// TIA Portal V18 export
FUNCTION_BLOCK "Capping_Station"   // FB1, LAD
TITLE = Description
{ S7_Optimized_Access := 'TRUE' }
VERSION : 0.1
// How to control and set capping station:
// 1) Start the machine
// 2) Use jog pos/neg in the capping station data block to rotate motor to read max and min value: ReadSensorMax and Read SensorMin. Based on these values update "SensorPosValMax..." and "SensorPosValMin..."
// 3) Move capping station using "MovingUP" and "MovingDOWN". The mechanism should stop top or bottom and confirm it with the change of the status "CSPositionUP" and "CSPositionDOWN". If it is constantly moving, it means that the value was not reached (too low for SensorPosValMin or too high for "SensorPosValMax").
// 
// IMPORTANT:
// - assembly of the mechanism needs to be the same, especially the position of the sensor
// - power supply for the sensor should be set to the exact voltage (5V) to provide repeteable readings
// 
// Things to implement:
// - Change sensor for limit switch
// - Improve mechanical design
// 
// E-STOP - always check!
// stored: AutoNumber true, IsIECCheckEnabled false, IsRetainMemResEnabled false, MemoryReserve 100, SetENOAutomatically false, UDAEnableTagReadback false
   VAR_INPUT
      ESTOP : Bool;
      SerialNumber : Int;
      CappingOption : Int;   // Send 1 to skip capping station
      MachineStart : Bool;
      CappingSensor : UInt;
      JogPOS : Bool;
      JogNEG : Bool;
      MoveRel : Bool;
      AxisXNotMoving : Bool;
      AxisYNotMoving : Bool;
      DoorSensor : Bool;
   END_VAR
   VAR_OUTPUT
      MovingUP : Bool;
      MovingDOWN : Bool;
      CSPositionUP : Bool;
      CSPositionDOWN : Bool;
      CSXYMotionLock : Bool;
      CappingPosition : UInt;
      MaintenanceNeeded : Bool;
   END_VAR
   VAR_IN_OUT
      CSMoveUP : Bool;
      CSMoveDOWN : Bool;
   END_VAR
   VAR
      MotionLockInternal : Bool;
      TimeSafety : Bool;
      SensorConversion : Real;
      SensorPosValMaxTrigger : UInt;
      SensorPosValMinTrigger : UInt;
      ReadSensorMax : UInt;   // Use jogging to read initial limit values
      ReadSensorMin : UInt := 10000;   // Use jogging to read initial limit values
      CountSinceON : DInt;
   END_VAR
   VAR RETAIN
      CountSinceNEW : DInt;
   END_VAR
   VAR
      MaintenanceMotionLockDisabled : Bool := true;
      SensorPosValMin { ExternalAccessible := 'False'; ExternalVisible := 'False'; ExternalWritable := 'False'} : UInt;   // 0; 14000; Machine 2009: 9000
      SensorPosValMax { ExternalAccessible := 'False'; ExternalVisible := 'False'; ExternalWritable := 'False'} : UInt;   // 6000; 21000; Machine 2009: 24500
      ScaleRangeMin { ExternalAccessible := 'False'; ExternalVisible := 'False'; ExternalWritable := 'False'} : UInt;   // 2009: 26000; 2008 20000;
      ScaleRangeMax { ExternalAccessible := 'False'; ExternalVisible := 'False'; ExternalWritable := 'False'} : UInt;   // 2009: 12000; 2008 4200;
   END_VAR
   VAR_TEMP
      JoggingPOSInternal : Bool;
      JoggingNEGInternal : Bool;
      CSPositionUPInternal : Bool;
      CSPositionDOWNInternal : Bool;
      MovingPermission : Bool;
   END_VAR
   VAR CONSTANT
      SensorPosValMax2008 : UInt := 15000;
      SensorPosValMax2009 : UInt := 24500;   // Armadillo 2009
      SensorPosValMax2010 : UInt := 17000;   // Armadillo 2010
      SensorPosValMax2011 : UInt := 13000;
      SensorPosValMax2012 : UInt := 14000;
      SensorPosValMin2008 : UInt := 5300;
      SensorPosValMin2009 : UInt := 9000;   // Armadillo 2009
      SensorPosValMin2010 : UInt := 4300;   // Armadillo 2010
      SensorPosValMin2011 : UInt := 4300;
      SensorPosValMin2012 : UInt := 4300;
      SensorPosTopMargin : UInt := 2000;   // 2000
      SensorPosBottomMargin : UInt := 2000;   // 2000
      ScaleRangeMax2008 : UInt := 18000;
      ScaleRangeMax2009 : UInt := 26000;
      ScaleRangeMax2010 : UInt := 18000;
      ScaleRangeMax2011 : UInt := 18000;
      ScaleRangeMax2012 : UInt := 18000;
      ScaleRangeMin2008 : UInt := 8000;
      ScaleRangeMin2009 : UInt := 8000;
      ScaleRangeMin2010 : UInt := 4200;
      ScaleRangeMin2011 : UInt := 8000;
      ScaleRangeMin2012 : UInt := 8000;
      MoveLength : DInt := 10000;   // microns
      MovementVelocity : Real := 90.0;   // 90
   END_VAR
   VAR_TEMP   // added for the SCL form of the ladder/FBD networks
      _w1 : Bool;
   END_VAR
BEGIN

REGION Network 1: Limit settings for different machines
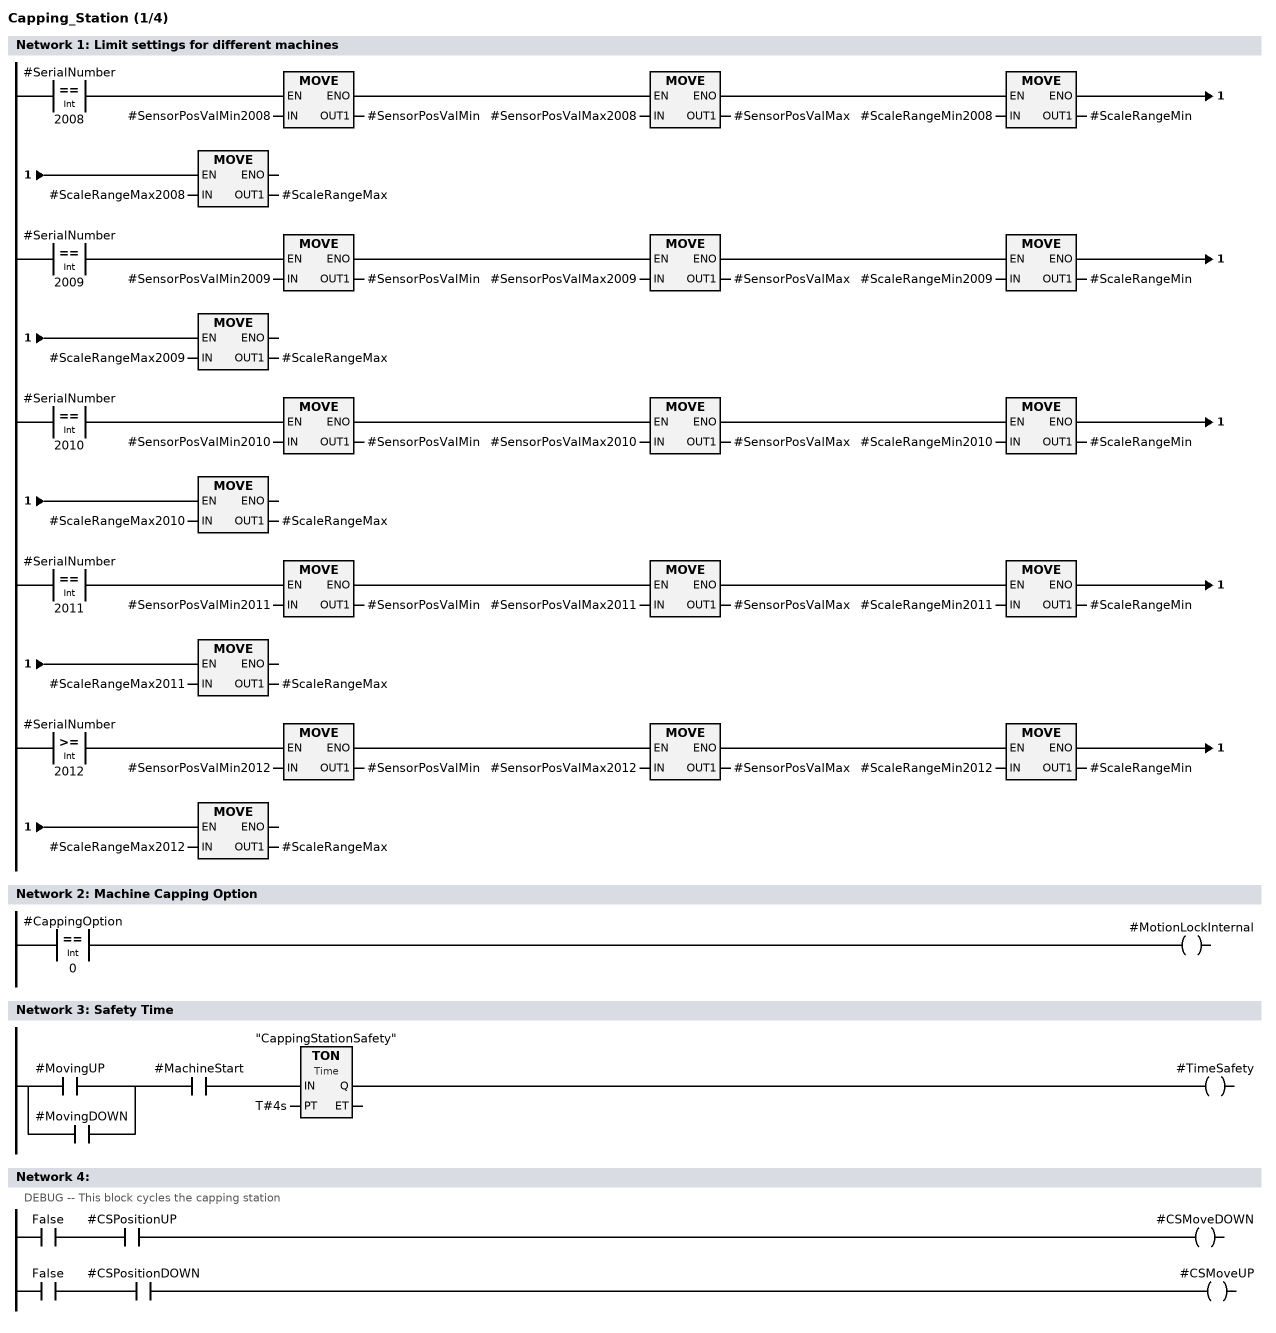
   RUNG wire#powerrail
      { S7_Templates := "SrcType := Int" } EQ_Contact(in1 := #SerialNumber, in2 := 2008)
      Move(in := #SensorPosValMin2008, out1 => #SensorPosValMin)
      Move(in := #SensorPosValMax2008, out1 => #SensorPosValMax)
      Move(in := #ScaleRangeMin2008, out1 => #ScaleRangeMin)
      Move(in := #ScaleRangeMax2008, out1 => #ScaleRangeMax)
   END_RUNG
   RUNG wire#powerrail
      { S7_Templates := "SrcType := Int" } EQ_Contact(in1 := #SerialNumber, in2 := 2009)
      Move(in := #SensorPosValMin2009, out1 => #SensorPosValMin)
      Move(in := #SensorPosValMax2009, out1 => #SensorPosValMax)
      Move(in := #ScaleRangeMin2009, out1 => #ScaleRangeMin)
      Move(in := #ScaleRangeMax2009, out1 => #ScaleRangeMax)
   END_RUNG
   RUNG wire#powerrail
      { S7_Templates := "SrcType := Int" } EQ_Contact(in1 := #SerialNumber, in2 := 2010)
      Move(in := #SensorPosValMin2010, out1 => #SensorPosValMin)
      Move(in := #SensorPosValMax2010, out1 => #SensorPosValMax)
      Move(in := #ScaleRangeMin2010, out1 => #ScaleRangeMin)
      Move(in := #ScaleRangeMax2010, out1 => #ScaleRangeMax)
   END_RUNG
   RUNG wire#powerrail
      { S7_Templates := "SrcType := Int" } EQ_Contact(in1 := #SerialNumber, in2 := 2011)
      Move(in := #SensorPosValMin2011, out1 => #SensorPosValMin)
      Move(in := #SensorPosValMax2011, out1 => #SensorPosValMax)
      Move(in := #ScaleRangeMin2011, out1 => #ScaleRangeMin)
      Move(in := #ScaleRangeMax2011, out1 => #ScaleRangeMax)
   END_RUNG
   RUNG wire#powerrail
      { S7_Templates := "SrcType := Int" } GE_Contact(in1 := #SerialNumber, in2 := 2012)
      Move(in := #SensorPosValMin2012, out1 => #SensorPosValMin)
      Move(in := #SensorPosValMax2012, out1 => #SensorPosValMax)
      Move(in := #ScaleRangeMin2012, out1 => #ScaleRangeMin)
      Move(in := #ScaleRangeMax2012, out1 => #ScaleRangeMax)
   END_RUNG
   // the same network as SCL:
   IF #SerialNumber = 2008 THEN
       #SensorPosValMin := #SensorPosValMin2008;
       #SensorPosValMax := #SensorPosValMax2008;
       #ScaleRangeMin := #ScaleRangeMin2008;
       #ScaleRangeMax := #ScaleRangeMax2008;
   END_IF;
   IF #SerialNumber = 2009 THEN
       #SensorPosValMin := #SensorPosValMin2009;
       #SensorPosValMax := #SensorPosValMax2009;
       #ScaleRangeMin := #ScaleRangeMin2009;
       #ScaleRangeMax := #ScaleRangeMax2009;
   END_IF;
   IF #SerialNumber = 2010 THEN
       #SensorPosValMin := #SensorPosValMin2010;
       #SensorPosValMax := #SensorPosValMax2010;
       #ScaleRangeMin := #ScaleRangeMin2010;
       #ScaleRangeMax := #ScaleRangeMax2010;
   END_IF;
   IF #SerialNumber = 2011 THEN
       #SensorPosValMin := #SensorPosValMin2011;
       #SensorPosValMax := #SensorPosValMax2011;
       #ScaleRangeMin := #ScaleRangeMin2011;
       #ScaleRangeMax := #ScaleRangeMax2011;
   END_IF;
   IF #SerialNumber >= 2012 THEN
       #SensorPosValMin := #SensorPosValMin2012;
       #SensorPosValMax := #SensorPosValMax2012;
       #ScaleRangeMin := #ScaleRangeMin2012;
       #ScaleRangeMax := #ScaleRangeMax2012;
   END_IF;
END_REGION

REGION Network 2: Machine Capping Option
   RUNG wire#powerrail
      { S7_Templates := "SrcType := Int" } EQ_Contact(in1 := #CappingOption, in2 := 0)
      Coil( #MotionLockInternal )
   END_RUNG
   // the same network as SCL:
   #MotionLockInternal := #CappingOption = 0;
END_REGION

REGION Network 3: Safety Time
   RUNG wire#powerrail
      Contact( #MovingUP )
      wire#w1
      Contact( #MachineStart )
      { S7_Templates := "time_type := Time" } "CappingStationSafety".TON(pt := T#4s, et =>)
      Coil( #TimeSafety )
   END_RUNG
   RUNG wire#powerrail
      Contact( #MovingDOWN )
   END_RUNG wire#w1
   // the same network as SCL:
   "CappingStationSafety".TON(IN := (#MovingUP OR #MovingDOWN) AND #MachineStart, PT := T#4s);
   #TimeSafety := "CappingStationSafety".Q;
END_REGION

REGION Network 4
   // DEBUG -- This block cycles the capping station
   RUNG wire#powerrail
      Contact( False )
      Contact( #CSPositionUP )
      Coil( #CSMoveDOWN )
   END_RUNG
   RUNG wire#powerrail
      Contact( False )
      Contact( #CSPositionDOWN )
      Coil( #CSMoveUP )
   END_RUNG
   // the same network as SCL:
   #CSMoveDOWN := False AND #CSPositionUP;
   #CSMoveUP := False AND #CSPositionDOWN;
END_REGION

REGION Network 5: Read Sensor Range
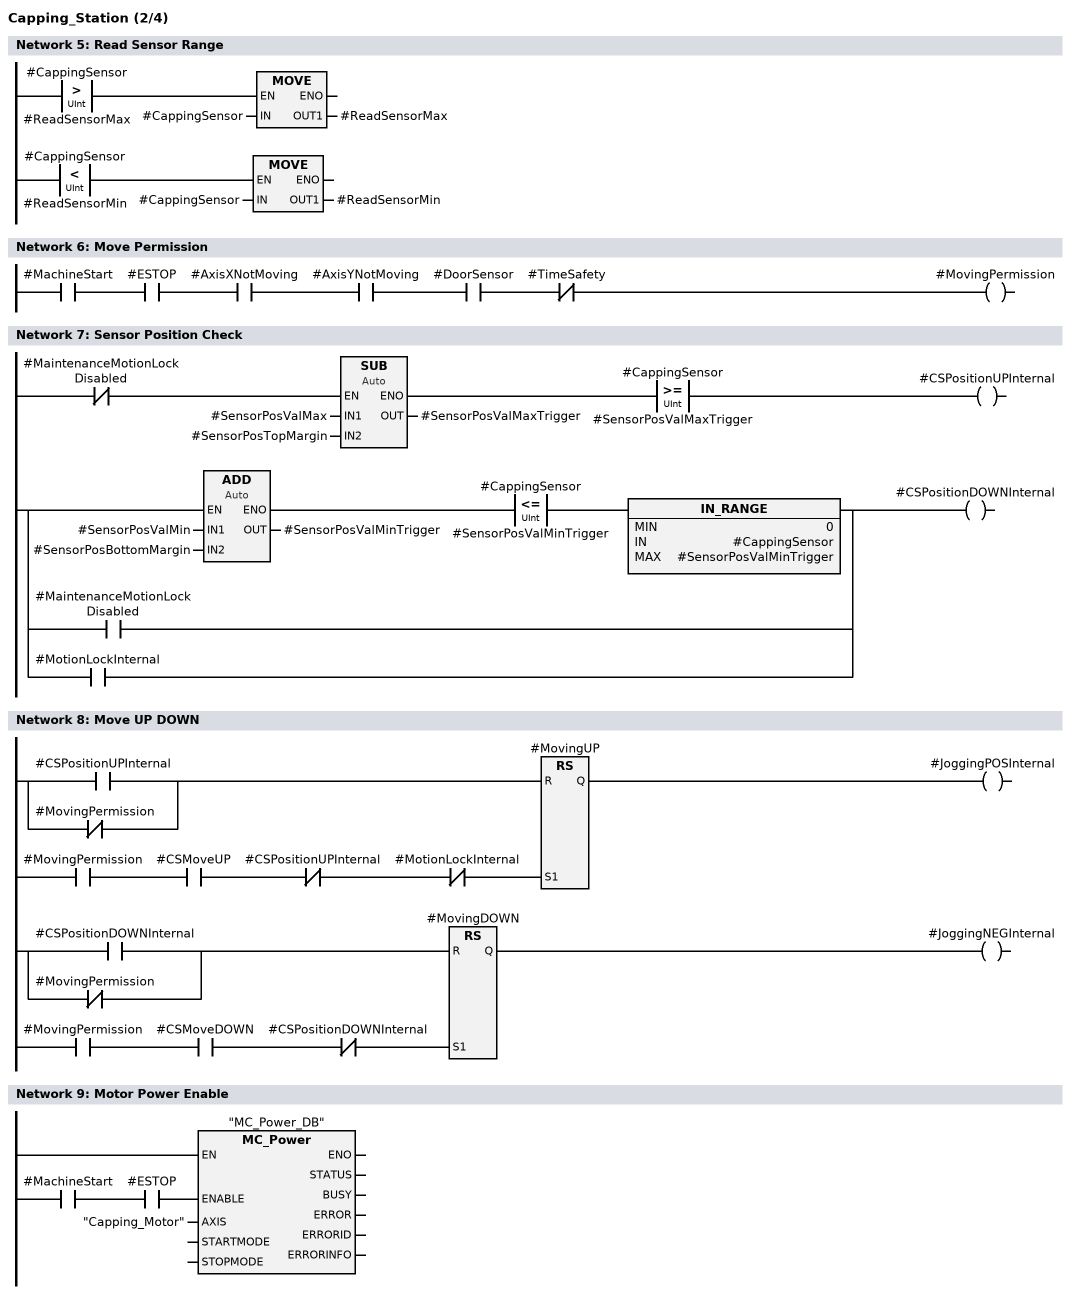
   RUNG wire#powerrail
      { S7_Templates := "SrcType := UInt" } GT_Contact(in1 := #CappingSensor, in2 := #ReadSensorMax)
      Move(in := #CappingSensor, out1 => #ReadSensorMax)
   END_RUNG
   RUNG wire#powerrail
      { S7_Templates := "SrcType := UInt" } LT_Contact(in1 := #CappingSensor, in2 := #ReadSensorMin)
      Move(in := #CappingSensor, out1 => #ReadSensorMin)
   END_RUNG
   // the same network as SCL:
   IF #CappingSensor > #ReadSensorMax THEN #ReadSensorMax := #CappingSensor; END_IF;
   IF #CappingSensor < #ReadSensorMin THEN #ReadSensorMin := #CappingSensor; END_IF;
END_REGION

REGION Network 6: Move Permission
   RUNG wire#powerrail
      Contact( #MachineStart )
      Contact( #ESTOP )
      Contact( #AxisXNotMoving )
      Contact( #AxisYNotMoving )
      Contact( #DoorSensor )
      I_Contact( #TimeSafety )
      Coil( #MovingPermission )
   END_RUNG
   // the same network as SCL:
   #MovingPermission := #MachineStart AND #ESTOP AND #AxisXNotMoving AND #AxisYNotMoving AND #DoorSensor AND NOT #TimeSafety;
END_REGION

REGION Network 7: Sensor Position Check
   RUNG wire#powerrail
      I_Contact( #MaintenanceMotionLockDisabled )
      Sub(in1 := #SensorPosValMax, in2 := #SensorPosTopMargin, out => #SensorPosValMaxTrigger)
      { S7_Templates := "SrcType := UInt" } GE_Contact(in1 := #CappingSensor, in2 := #SensorPosValMaxTrigger)
      Coil( #CSPositionUPInternal )
   END_RUNG
   RUNG wire#powerrail
      Add(in1 := #SensorPosValMin, in2 := #SensorPosBottomMargin, out => #SensorPosValMinTrigger)
      { S7_Templates := "SrcType := UInt" } LE_Contact(in1 := #CappingSensor, in2 := #SensorPosValMinTrigger)
      { S7_Templates := "SrcType := UInt" } InRange(min := 0, in := #CappingSensor, max := #SensorPosValMinTrigger)
      wire#w1
      Coil( #CSPositionDOWNInternal )
   END_RUNG
   RUNG wire#powerrail
      Contact( #MaintenanceMotionLockDisabled )
   END_RUNG wire#w1
   RUNG wire#powerrail
      Contact( #MotionLockInternal )
   END_RUNG wire#w1
   // the same network as SCL:
   #_w1 := NOT #MaintenanceMotionLockDisabled;
   IF #_w1 THEN #SensorPosValMaxTrigger := #SensorPosValMax - #SensorPosTopMargin; END_IF;
   #CSPositionUPInternal := #_w1 AND (#CappingSensor >= #SensorPosValMaxTrigger);
   #SensorPosValMinTrigger := #SensorPosValMin + #SensorPosBottomMargin;
   #CSPositionDOWNInternal := ((#CappingSensor <= #SensorPosValMinTrigger) AND (0 <= #CappingSensor) AND (#CappingSensor <= #SensorPosValMinTrigger)) OR #MaintenanceMotionLockDisabled OR #MotionLockInternal;
END_REGION

REGION Network 8: Move UP DOWN
   RUNG wire#powerrail
      Contact( #CSPositionUPInternal )
      wire#w1
      S_RS(operand := #MovingUP, s1 := wire#w2)
      Coil( #JoggingPOSInternal )
   END_RUNG
   RUNG wire#powerrail
      I_Contact( #MovingPermission )
   END_RUNG wire#w1
   RUNG wire#powerrail
      Contact( #MovingPermission )
      Contact( #CSMoveUP )
      I_Contact( #CSPositionUPInternal )
      I_Contact( #MotionLockInternal )
   END_RUNG wire#w2
   RUNG wire#powerrail
      Contact( #CSPositionDOWNInternal )
      wire#w3
      S_RS(operand := #MovingDOWN, s1 := wire#w4)
      Coil( #JoggingNEGInternal )
   END_RUNG
   RUNG wire#powerrail
      I_Contact( #MovingPermission )
   END_RUNG wire#w3
   RUNG wire#powerrail
      Contact( #MovingPermission )
      Contact( #CSMoveDOWN )
      I_Contact( #CSPositionDOWNInternal )
   END_RUNG wire#w4
   // the same network as SCL:
   IF #CSPositionUPInternal OR NOT #MovingPermission THEN
       #MovingUP := FALSE;   // RS flip-flop
   END_IF;
   IF #MovingPermission AND #CSMoveUP AND NOT #CSPositionUPInternal AND NOT #MotionLockInternal THEN
       #MovingUP := TRUE;
   END_IF;
   #JoggingPOSInternal := #MovingUP;
   IF #CSPositionDOWNInternal OR NOT #MovingPermission THEN
       #MovingDOWN := FALSE;   // RS flip-flop
   END_IF;
   IF #MovingPermission AND #CSMoveDOWN AND NOT #CSPositionDOWNInternal THEN #MovingDOWN := TRUE; END_IF;
   #JoggingNEGInternal := #MovingDOWN;
END_REGION

REGION Network 9: Motor Power Enable
   RUNG wire#powerrail
      "MC_Power_DB".MC_Power(Enable := wire#w1, Axis := "Capping_Motor", StartMode :=, StopMode :=, Status =>, Busy =>, Error =>, ErrorID =>, ErrorInfo =>)
   END_RUNG
   RUNG wire#powerrail
      Contact( #MachineStart )
      Contact( #ESTOP )
   END_RUNG wire#w1
   // the same network as SCL:
   "MC_Power_DB"(Enable := #MachineStart AND #ESTOP, Axis := "Capping_Motor");   // MC_Power
END_REGION

REGION Network 10: Move Jog
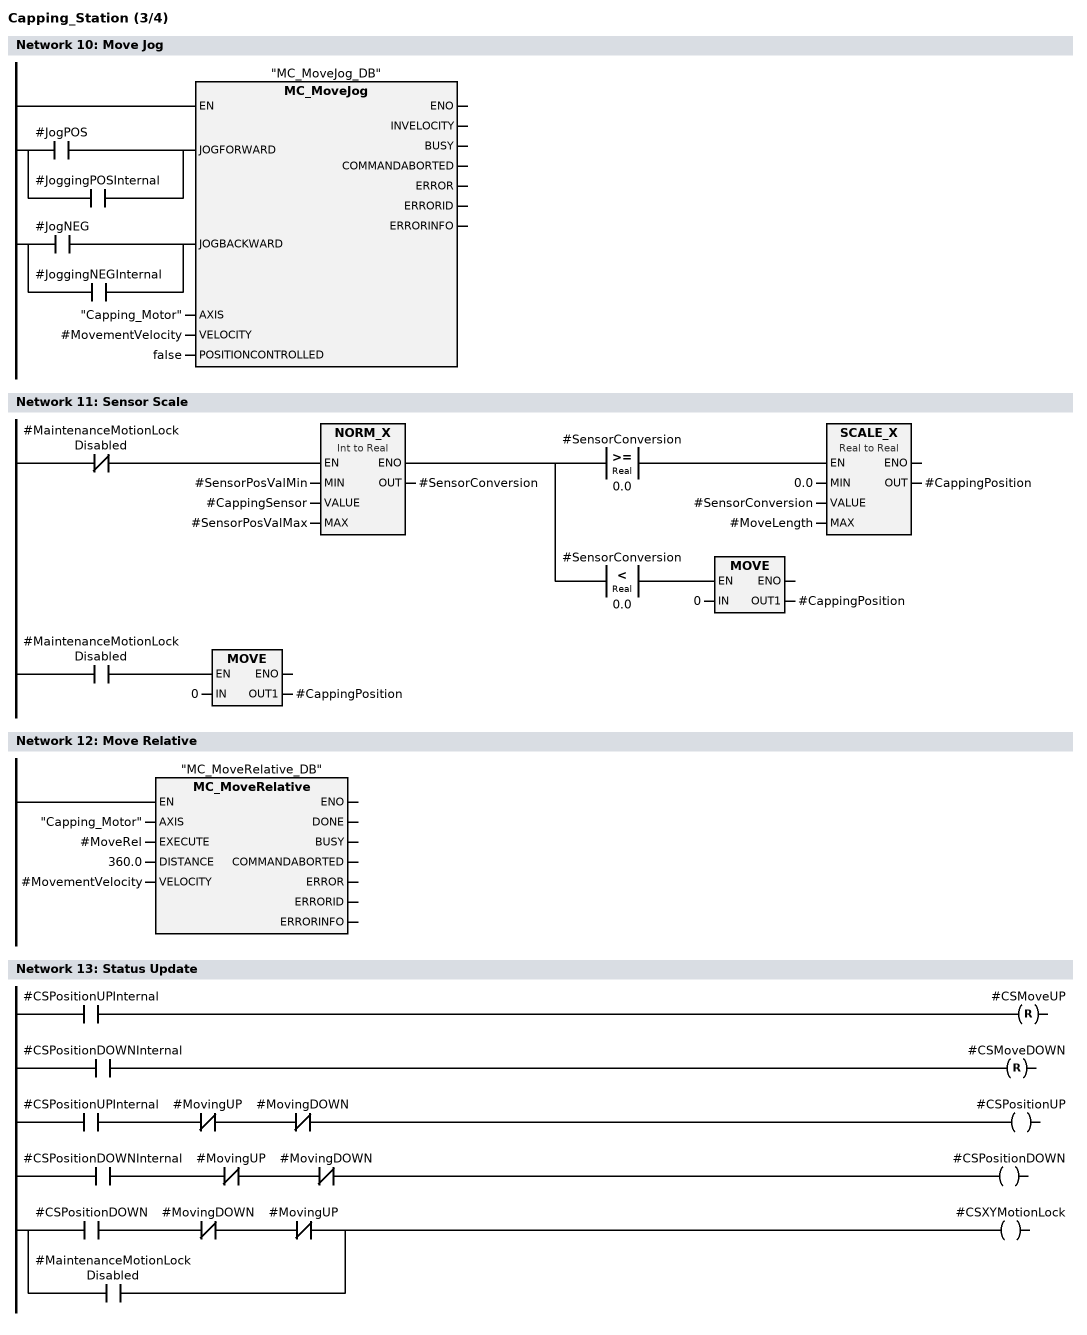
   RUNG wire#powerrail
      "MC_MoveJog_DB".MC_MoveJog(JogForward := wire#w1, JogBackward := wire#w2, Axis := "Capping_Motor", Velocity := #MovementVelocity, PositionControlled := false, InVelocity =>, Busy =>, CommandAborted =>, Error =>, ErrorID =>, ErrorInfo =>)
   END_RUNG
   RUNG wire#powerrail
      Contact( #JogPOS )
   END_RUNG wire#w1
   RUNG wire#powerrail
      Contact( #JoggingPOSInternal )
   END_RUNG wire#w1
   RUNG wire#powerrail
      Contact( #JogNEG )
   END_RUNG wire#w2
   RUNG wire#powerrail
      Contact( #JoggingNEGInternal )
   END_RUNG wire#w2
   // the same network as SCL:
   "MC_MoveJog_DB"(JogForward := #JogPOS OR #JoggingPOSInternal,   // MC_MoveJog
                   JogBackward := #JogNEG OR #JoggingNEGInternal,
                   Axis := "Capping_Motor",
                   Velocity := #MovementVelocity,
                   PositionControlled := false);
END_REGION

REGION Network 11: Sensor Scale
   RUNG wire#powerrail
      I_Contact( #MaintenanceMotionLockDisabled )
      { S7_Templates := "[SrcType := Int, DestType := Real]" } Normalize(min := #SensorPosValMin, value := #CappingSensor, max := #SensorPosValMax, out => #SensorConversion)
      wire#w1
      { S7_Templates := "SrcType := Real" } GE_Contact(in1 := #SensorConversion, in2 := 0.0)
      { S7_Templates := "[SrcType := Real, DestType := Real]" } Scale(min := 0.0, value := #SensorConversion, max := #MoveLength, out => #CappingPosition)
   END_RUNG
   RUNG wire#w1
      { S7_Templates := "SrcType := Real" } LT_Contact(in1 := #SensorConversion, in2 := 0.0)
      Move(in := 0, out1 => #CappingPosition)
   END_RUNG
   RUNG wire#powerrail
      Contact( #MaintenanceMotionLockDisabled )
      Move(in := 0, out1 => #CappingPosition)
   END_RUNG
   // the same network as SCL:
   #_w1 := NOT #MaintenanceMotionLockDisabled;
   IF #_w1 THEN
       #SensorConversion := NORM_X(MIN := #SensorPosValMin, VALUE := #CappingSensor, MAX := #SensorPosValMax);
   END_IF;
   IF #_w1 AND (#SensorConversion >= 0.0) THEN
       #CappingPosition := SCALE_X(MIN := 0.0, VALUE := #SensorConversion, MAX := #MoveLength);
   END_IF;
   IF #_w1 AND (#SensorConversion < 0.0) THEN #CappingPosition := 0; END_IF;
   IF #MaintenanceMotionLockDisabled THEN #CappingPosition := 0; END_IF;
END_REGION

REGION Network 12: Move Relative
   RUNG wire#powerrail
      "MC_MoveRelative_DB".MC_MoveRelative(Axis := "Capping_Motor", Execute := #MoveRel, Distance := 360.0, Velocity := #MovementVelocity, Done =>, Busy =>, CommandAborted =>, Error =>, ErrorID =>, ErrorInfo =>)
   END_RUNG
   // the same network as SCL:
   "MC_MoveRelative_DB"(Axis := "Capping_Motor",   // MC_MoveRelative
                        Execute := #MoveRel,
                        Distance := 360.0,
                        Velocity := #MovementVelocity);
END_REGION

REGION Network 13: Status Update
   RUNG wire#powerrail
      Contact( #CSPositionUPInternal )
      R_Coil( #CSMoveUP )
   END_RUNG
   RUNG wire#powerrail
      Contact( #CSPositionDOWNInternal )
      R_Coil( #CSMoveDOWN )
   END_RUNG
   RUNG wire#powerrail
      Contact( #CSPositionUPInternal )
      I_Contact( #MovingUP )
      I_Contact( #MovingDOWN )
      Coil( #CSPositionUP )
   END_RUNG
   RUNG wire#powerrail
      Contact( #CSPositionDOWNInternal )
      I_Contact( #MovingUP )
      I_Contact( #MovingDOWN )
      Coil( #CSPositionDOWN )
   END_RUNG
   RUNG wire#powerrail
      Contact( #CSPositionDOWN )
      I_Contact( #MovingDOWN )
      I_Contact( #MovingUP )
      wire#w1
      Coil( #CSXYMotionLock )
   END_RUNG
   RUNG wire#powerrail
      Contact( #MaintenanceMotionLockDisabled )
   END_RUNG wire#w1
   // the same network as SCL:
   IF #CSPositionUPInternal THEN #CSMoveUP := FALSE; END_IF;
   IF #CSPositionDOWNInternal THEN #CSMoveDOWN := FALSE; END_IF;
   #CSPositionUP := #CSPositionUPInternal AND NOT #MovingUP AND NOT #MovingDOWN;
   #CSPositionDOWN := #CSPositionDOWNInternal AND NOT #MovingUP AND NOT #MovingDOWN;
   #CSXYMotionLock := (#CSPositionDOWN AND NOT #MovingDOWN AND NOT #MovingUP) OR #MaintenanceMotionLockDisabled;
END_REGION

REGION Network 14: Moves counter
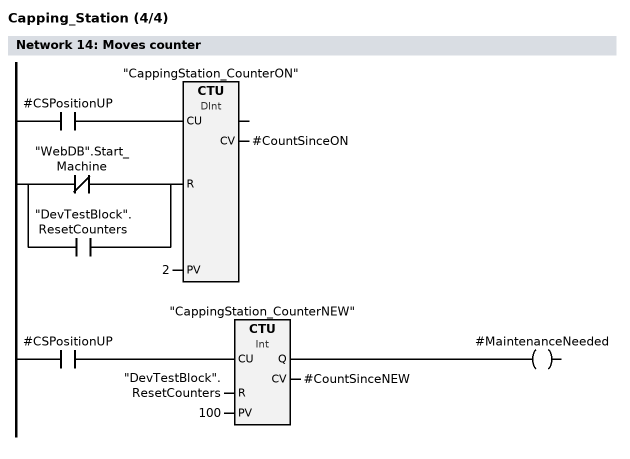
   RUNG wire#powerrail
      Contact( #CSPositionUP )
      { S7_Templates := "value_type := DInt" } "CappingStation_CounterON".CTU(r := wire#w1, pv := 2, cv => #CountSinceON)
   END_RUNG
   RUNG wire#powerrail
      I_Contact( "WebDB".Start_Machine )
   END_RUNG wire#w1
   RUNG wire#powerrail
      Contact( "DevTestBlock".ResetCounters )
   END_RUNG wire#w1
   RUNG wire#powerrail
      Contact( #CSPositionUP )
      { S7_Templates := "value_type := Int" } "CappingStation_CounterNEW".CTU(r := "DevTestBlock".ResetCounters, pv := 100, cv => #CountSinceNEW)
      Coil( #MaintenanceNeeded )
   END_RUNG
   // the same network as SCL:
   "CappingStation_CounterON".CTU(CU := #CSPositionUP,
                           R := NOT "WebDB".Start_Machine OR "DevTestBlock".ResetCounters,
                           PV := 2,
                           CV => #CountSinceON);
   "CappingStation_CounterNEW".CTU(CU := #CSPositionUP,
                           R := "DevTestBlock".ResetCounters,
                           PV := 100,
                           CV => #CountSinceNEW);
   #MaintenanceNeeded := "CappingStation_CounterNEW".Q;
END_REGION
END_FUNCTION_BLOCK
